FUNCTION_BLOCK FB_Plant
VAR_INPUT
	bAuto_IN : BOOL;
	bManual_IN :BOOL;
	
	bStart_IN : BOOL;
	bStop_IN :BOOL;
	bReset_IN : BOOL;
	bEmgStop_IN : BOOL;
	
END_VAR

VAR_OUTPUT
	bAuto_OUT :BOOL;
	bManual_OUT :BOOL;
	
	bStarted :BOOL;
	bStopped : BOOL;
END_VAR

VAR_IN_OUT
	PlantCtrl : Plant_CTRL;
END_VAR

VAR
END_VAR
VAR // added by the converter: edge detectors and wires of the graphical bodies
    _w1, _w2 : BOOL;
END_VAR

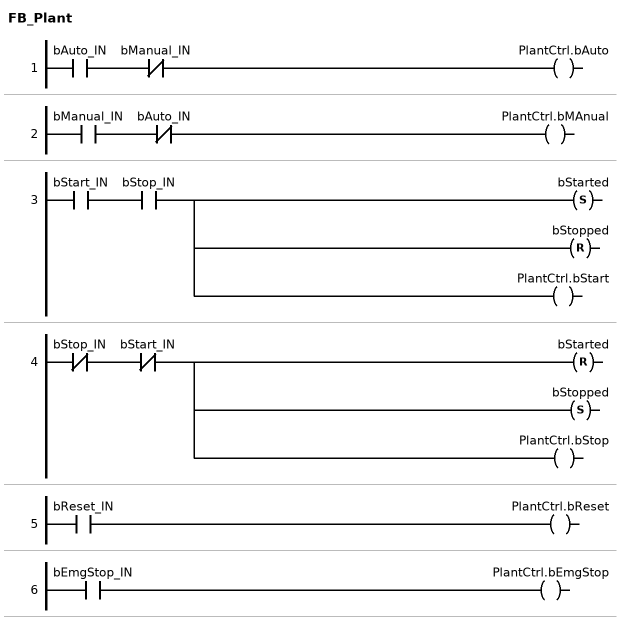
// NETWORK 1
PlantCtrl.bAuto := bAuto_IN AND NOT bManual_IN;

// NETWORK 2
PlantCtrl.bMAnual := bManual_IN AND NOT bAuto_IN;

// NETWORK 3
_w1 := bStart_IN AND bStop_IN;
bStarted S= _w1;
bStopped R= _w1;
PlantCtrl.bStart := _w1;

// NETWORK 4
_w2 := NOT bStop_IN AND NOT bStart_IN;
bStarted R= _w2;
bStopped S= _w2;
PlantCtrl.bStop := _w2;

// NETWORK 5
PlantCtrl.bReset := bReset_IN;

// NETWORK 6
PlantCtrl.bEmgStop := bEmgStop_IN;

END_FUNCTION_BLOCK

(* stored: Version 1.1.0.1, ProductVersion 3.1.4024.13
   POU FB_Plant: Id {cac6cf26-aacf-4de4-88aa-5821726ce651}, SpecialFunc None *)
